FUNCTION_BLOCK Buffer

VAR CONSTANT
	AxesMaxAmount : USINT := 6;
	PosMaxAmount : USINT := 10;
END_VAR

VAR
	bInit : BOOL := TRUE;
	POS_STORAGE : ARRAY [1..PosMaxAmount] OF ARRAY [1..AxesMaxAmount] OF LREAL;
	InCommand : Motion_Command_Input;
END_VAR



InCommand.StartPos := InCommand.StartPOS;

END_FUNCTION_BLOCK

(* stored: Version 1.1.0.1, ProductVersion 3.1.4024.13
   POU Buffer: Id {148c26d4-7097-4286-a9e7-ba4d69266572}, SpecialFunc None *)
